FUNCTION_BLOCK FB_Gear
VAR_IN_OUT
	stGear:ST_Gear;
	AxisRefMaster:AXIS_REF;
	AxisRefSlave:AXIS_REF;
	stSystem:ST_System;
//	arrfbSetAlarm: ARRAY[1..3] OF FB_SetError;
END_VAR
VAR_INPUT
	inChannelid:INT;
END_VAR
VAR
	fbGearIn:MC_GearIn;
	fbGearInDyn:MC_GearInDyn;
	fbGearout:MC_GearOut;
	fbGearoutTrig:R_TRIG;
	arrfbSetAlarm: ARRAY[1..3] OF FB_SetError;
	i:UINT;
	statr: BOOL;
END_VAR

fbGearInDyn(
	Master:= AxisRefMaster, 
	Slave:= AxisRefSlave, 
	Enable:= stGear.bGearIn(*arstGear[2].bGearIn*), 
	GearRatio:=stGear.rRatioNumerator, 
	Acceleration:= , 
	Deceleration:= , 
	Jerk:= , 
	BufferMode:= , 
	Options:= , 
	InGear=> , 
	Busy=> , 
	Active=> , 
	CommandAborted=> , 
	Error=> stGear.bError, 
	ErrorID=> );
//fbGearIn(
//	Master:= stGear.AxisRefMaster, 
//	Slave:= stGear.AxisRefSlave, 
//	Execute:= stGear.bGearIn, 
//	RatioNumerator:= stGear.rRatioNumerator, 
//	RatioDenominator:= stGear.uiRatioDenominator, 
//	Acceleration:= , 
//	Deceleration:=, 
//	Jerk:= , 
//	BufferMode:= , 
//	Options:= , 
//	InGear=> , 
//	Busy=> , 
//	Active=> , 
//	CommandAborted=> , 
//	Error=> stGear.bError, 
//	ErrorID=> );
stGear.bInSyncing:=AxisRefSlave.Status.Coupled;
fbGearout(
	Slave:=  AxisRefSlave(*stGear.AxisRefSlave*) , 
	Execute:= stGear.bGearOut , 
	Options:= , 
	Done=> stGear.bnoInSyncing, 
	Busy=> , 
	Error=> stGear.bError, 
	ErrorID=> );
//fbGearoutTrig(CLK:=fbGearout.Done , Q=> );
//	IF fbGearoutTrig.Q THEN
//		stGear.bGearin:=FALSE;
//	END_IF
IF fbGearIn.Error THEN
	stGear.bError:=TRUE;
	stGear.arErrorID[1]:=TRUE;
//ELSIF fbGearInPos.Error THEN
	//stGear.arErrorID[2]:=TRUE;
ELSIF fbGearout.Error THEN
	stGear.bError:=TRUE;
	stGear.arErrorID[2]:=TRUE;
END_IF
// 耦合报错
arrfbSetAlarm[1](
	bEnable:= TRUE, 
	iErrorID:= 80+3*(inChannelid-1), 
	bExecute:= stGear.arErrorID[1], 
	bReset:= stSystem.bReset, 
	strErrorInfoEN:= 'Gear_in Alm', 
	wstrErrorInfoCN:="耦合错误" , 
	enumErrorClass:= 6, 
    );
// 耦合报错
arrfbSetAlarm[3](
	bEnable:= TRUE, 
	iErrorID:= 80+3*(inChannelid-1)+2, 
	bExecute:= stGear.arErrorID[3], 
	bReset:= stSystem.bReset, 
	strErrorInfoEN:= 'Gear_in Alm', 
	wstrErrorInfoCN:=" 解耦错误" , 
	enumErrorClass:= 6, 
    );
IF stSystem.bReset THEN
	stGear.bError:=FALSE;
	FOR i:=1 TO 2 BY 1 DO 
	   stGear.arErrorID[i]:=FALSE;
    END_FOR
END_IF

END_FUNCTION_BLOCK

(* stored: Version 1.1.0.1, ProductVersion 3.1.4024.12
   POU FB_Gear: Id {34eee4ab-e82e-41ce-bacf-9b80f0e79f97}, SpecialFunc None *)
